// TIA Portal V20 export
VAR_GLOBAL   // PLC tag table "IO_Device_PCL_Centralilze_PLC_Functinal_Test_2"
   In_Test_Parameters AT %I100.0 : "IO_Device_Test_Parameters";
   Out_Functinal_Test AT %Q100.0 : "IO_Device_Functinal_Test";
END_VAR
